{attribute 'qualified_only'}
{attribute 'strict'}
TYPE eActor :
(
	Human 			:= 0,
	Robot			:= 1,
	RemoteSystem	:= 2
);
END_TYPE

(* stored: Version 1.1.0.1, ProductVersion 3.1.4024.12
   EnumerationTextList eActorType: Id {7c315ced-fc40-402b-8895-601deeec7cfe} *)
